{attribute 'qualified_only'}
VAR_GLOBAL
	Encoder1NetCounts : LINT; 
	Encoder1Degrees : REAL; 
END_VAR

(* stored: Version 1.1.0.1, ProductVersion 3.1.4024.12
   GVL GVL: Id {d207ee37-d2d8-410e-b2c4-724ae4b38d12} *)
